{attribute 'linkalways'} 
{attribute 'no_explicit_call' := 'This FB is a CLASS and must be accessed using methods or properties'}
{attribute 'enable_dynamic_creation'}
FUNCTION_BLOCK EventHandlerItem EXTENDS Disposable IMPLEMENTS I_EventHandlerItem
VAR
	handler : I_EventHandler;
	_next : I_EventHandlerItem;
	_previous : I_EventHandlerItem;
END_VAR

METHOD PUBLIC Emit
VAR_INPUT
	Event : I_Event;
END_VAR
IF handler = 0 THEN
	RETURN;
END_IF

handler.HandleEvent(Event);
END_METHOD

METHOD EqualTo : BOOL
VAR_INPUT
	Handler : I_EventHandler;
END_VAR
EqualTo := THIS^.handler = Handler;
END_METHOD

METHOD FB_init : BOOL
VAR_INPUT
	bInitRetains : BOOL; // if TRUE, the retain variables are initialized (warm start / cold start)
	bInCopyCode : BOOL;  // if TRUE, the instance afterwards gets moved into the copy code (online change)
	Handler : I_EventHandler;
END_VAR
THIS^.handler := Handler;
END_METHOD

PROPERTY PUBLIC Next : I_EventHandlerItem
GET
Next := _next;
END_GET
SET
_next := Next;
END_SET
END_PROPERTY

METHOD PROTECTED OnDispose : BOOL
VAR_INPUT
	CalledExplicitly : BOOL;
END_VAR
// no other action needed
END_METHOD

PROPERTY PUBLIC Previous : I_EventHandlerItem
GET
Previous := _previous;
END_GET
SET
_previous := Previous;
END_SET
END_PROPERTY

END_FUNCTION_BLOCK

(* stored: Version 1.1.0.1, ProductVersion 3.1.4024.12
   POU EventHandlerItem: Id {663e3b97-05f1-00d9-21da-631d87d26eb9}, SpecialFunc None
   Folder Constructor: Id {7dd57d77-72d8-08b5-38c9-1fbebb7d8bed}
   Folder Protected: Id {d04a09b8-32c0-4d76-99ad-06262aec8ec2}
   Method Emit: Id {866eecf0-8116-015b-1dbb-47d7acd4d5e9}
   Method EqualTo: Id {0b7f4115-028c-0538-2e49-fc943848d717}
   Method FB_init: Id {05c029f5-291d-0e89-2a33-46bfdf5d0772}
   Property Next: Id {7c3a79d8-d51d-0b55-15cc-435911325a3c}
   Get Get: Id {387e05e0-8ff9-0726-1858-78b4668a0f4a}
   Set Set: Id {3a3150bf-b990-07b5-07a2-0fd0d28488c4}
   Method OnDispose: Id {bcd6bdb2-5daf-4b22-9f57-b784336d862d}
   Property Previous: Id {084ead29-15f0-0aa5-3c19-3f650ca0185f}
   Get Get: Id {cd2fabec-7383-0bb3-1699-4aab956b206c}
   Set Set: Id {35ee9d53-d6e4-0977-28aa-df5a8214dc49} *)
